PROGRAM SerialTxRx
VAR
END_VAR

M3SelectorA.SerialComm();
M3SelectorB.SerialComm();
M3SelectorC.SerialComm();
M3SelectorD.SerialComm();

PCMA.SerialComm();
PCMB.SerialComm();
PCMC.SerialComm();
PCMD.SerialComm();

END_PROGRAM

(* stored: Version 1.1.0.1, ProductVersion 3.1.4024.12
   POU SerialTxRx: Id {9fdbe883-e083-4b63-a863-4d2c242a797c}, SpecialFunc None *)
